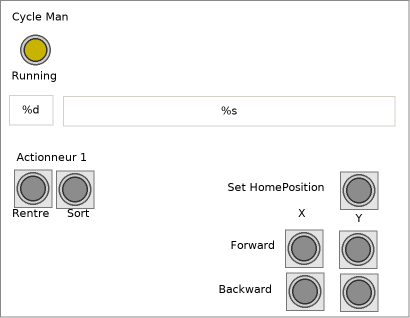
VISUALIZATION VisuManual  // 410x318
    Label (9,2 159x30), "Cycle Man"
    Label (5,61 59x30), "Running"
    Lamp1 (17,32 37x36), variable: fbCycleMan.xBusy, style: Lamp-Lamp1-Yellow
    PushSwitch (14,167 38x43), variable: stIO.stIn.xManualAct1GoIn, behaviour: TAP, style: Switch-PushSwitch-Gray
    PushSwitch (56,168 38x43), variable: stIO.stIn.xManualAct1GoOut, behaviour: TAP, style: Switch-PushSwitch-Gray
    Label (0,199 102x29), "Rentre Sort"
    Label (1,143 102x29), "Actionneur 1"
    Label (306,201 102x29)
    Textfield (63,96 332x30), "%s", text variable: fbCycleMan.fbEtape.sMess
    Textfield (9,95 44x30), "%d", text variable: fbCycleMan.iEtape
    Label (-2,287 155x29)
    Group (179,169 199x145)
        Label (2,62 97x29), "Forward", invisible if: fbCycleInit.iEtape<>500
        Label (0,106 96x29), "Backward", invisible if: fbCycleInit.iEtape<>500
        Group (46,0 153x145)
            PushSwitch (115,0 38x43), variable: stIO.stIn.xSetHomePos, invisible if: fbCycleInit.iEtape<>500, behaviour: TAP, style: Switch-PushSwitch-Gray
            Label (0,4 102x29), "Set HomePosition", invisible if: fbCycleInit.iEtape<>500
            PushSwitch (60,58 38x43), variable: stIO.stIn.xJogXForward, invisible if: fbCycleInit.iEtape<>500, behaviour: TAP, style: Switch-PushSwitch-Gray
            PushSwitch (115,102 38x43), variable: stIO.stIn.xJogYBackward, invisible if: fbCycleInit.iEtape<>500, behaviour: TAP, style: Switch-PushSwitch-Gray
            PushSwitch (114,59 38x43), variable: stIO.stIn.xJogYForward, invisible if: fbCycleInit.iEtape<>500, behaviour: TAP, style: Switch-PushSwitch-Gray
            PushSwitch (61,101 38x43), variable: stIO.stIn.xJogXBackward, invisible if: fbCycleInit.iEtape<>500, behaviour: TAP, style: Switch-PushSwitch-Gray
            Label (60,30 34x29), "X", invisible if: fbCycleInit.iEtape<>500
            Label (117,35 34x29), "Y", invisible if: fbCycleInit.iEtape<>500
END_VISUALIZATION

(* stored: Version 1.1.0.1, ProductVersion 3.1.4020.12
   Visu VisuManual: Id {f28ef4db-7197-4f06-b587-d328527c7bba} *)
